(*
    Determine whether a pump attached to the inlet of a roughing pump is safe to open.

    Return true, signaling it is safe to open when the roughing pump is confirmed to be working.
*)

FUNCTION F_RoughPumpInlet_ILK : BOOL
VAR_INPUT
    ScrollPump	:	ST_RoughPump;
END_VAR
VAR
END_VAR


F_RoughPumpInlet_ILK := (ScrollPump.eState = pumpRUNNING); (* Confirm that the roughing pump is running before opening the valve *)

END_FUNCTION

(* stored: Version 1.1.0.1
   POU F_RoughPumpInlet_ILK: Id {25dfe2f9-c6c4-41b1-9216-615302b27fca}, SpecialFunc None *)
